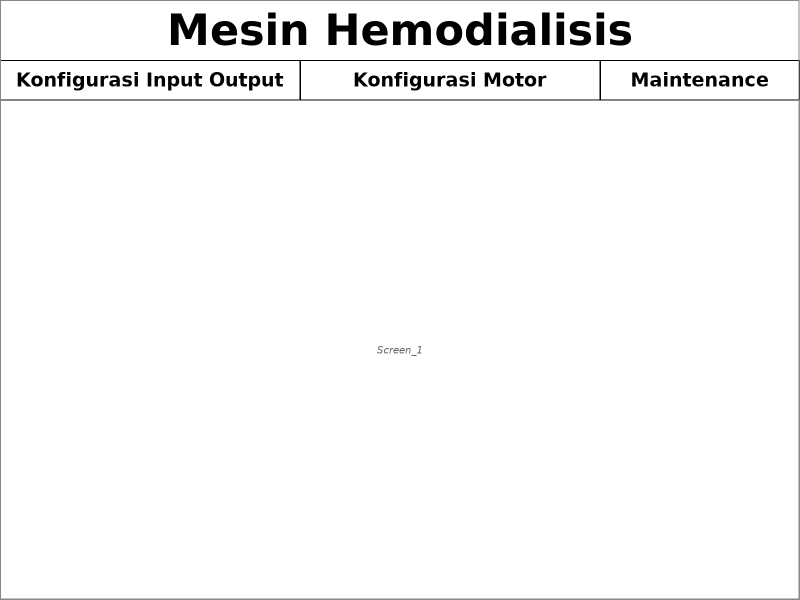
VISUALIZATION Main_Screen  // 800x600
    Label (0,0 800x60), "Mesin Hemodialisis"
    Rectangle (0,60 300x40), "Konfigurasi Input Output"
        OnMouseClick: FrameSelectionChange Selection=SelectedFrame=429c0b64-bdc9-449d-b1bd-91a074b8e2d9, GlobSel=AssignType=Directly, SelType=Locally
    Rectangle (300,60 300x40), "Konfigurasi Motor"
        OnMouseClick: FrameSelectionChange Selection=SelectedFrame=429c0b64-bdc9-449d-b1bd-91a074b8e2d9, Selection=1, GlobSel=AssignType=Directly, SelType=Locally
    Rectangle (600,60 200x40), "Maintenance"
        OnMouseClick: FrameSelectionChange Selection=SelectedFrame=429c0b64-bdc9-449d-b1bd-91a074b8e2d9, Selection=2, GlobSel=AssignType=Directly, SelType=Locally
    Frame (0,100 800x500)
        shows Screen_1()
        shows Screen_2()
        shows Screen_3()
END_VISUALIZATION

(* stored: Version 1.1.0.1, ProductVersion 3.1.4024.12
   Visu Main_Screen: Id {b3c179e4-dc64-4530-861f-8b1a0e139a76} *)
